// TIA Portal V19 export
DATA_BLOCK "EmNodes"   // DB146
// Global DB for the data exchange between the module levels (Between Unit and EM or EM and CM)
// stored: Access Published, MemoryReserve 100, Namespace Unit
   VAR
      unitStatus { ExternalWritable := 'False'} : "LAF_typeUnitStatus";   // Status of the unit
      emFeedback { ExternalWritable := 'False'} : Array[0.._.NO_OF_EMs] of "LUC_typeEmFeedback";   // Status of the individual equipment modules
      emRelations { ExternalWritable := 'False'} : Struct   // This is an example
         EM0 : Struct
            readyToReceive : Bool;
            readyToDeliver : Bool;
         END_STRUCT;
         EM1 : Struct
            readyToReceive : Bool;
            readyToDeliver : Bool;
         END_STRUCT;
         EM2 : Struct
            readyToReceive : Bool;
            readyToDeliver : Bool;
         END_STRUCT;
      END_STRUCT;
      signalStack { ExternalWritable := 'False'} : "LUC_typeSignalStackByBool";
   END_VAR
BEGIN
END_DATA_BLOCK
